FUNCTION_BLOCK FB_EmpujarPlato_SFC

VAR_IN_OUT
	   TpoEmpujadorAvanza: TIME;
END_VAR

VAR_INPUT
    // SFC-Flags
    SFCPause: BOOL;
    SFCReset: BOOL;
    
    // Indicadores de sincronizacion
    Ack: BOOL := TRUE;
    Execute: BOOL;
    
    
    // Entradas
   PlatoEmpujadorDetras : BOOL;
END_VAR
VAR_OUTPUT
    // Indicadores de sincronizacion
    Done: BOOL;
    Ready: BOOL;
    
    // Salidas
    PlatoEmpujadorAvanza : BOOL;
	PlatoRetenedorAtras : BOOL;
END_VAR
VAR
END_VAR

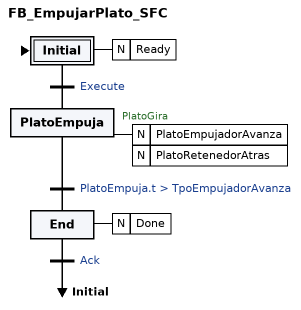
INITIAL_STEP Initial:
    Ready(N);
END_STEP
TRANSITION FROM Initial TO PlatoEmpuja
    := Execute;
END_TRANSITION
// PlatoGira
STEP PlatoEmpuja:
    PlatoEmpujadorAvanza(N);
    PlatoRetenedorAtras(N);
END_STEP
TRANSITION FROM PlatoEmpuja TO End
    := PlatoEmpuja.t > TpoEmpujadorAvanza;
END_TRANSITION
STEP End:
    Done(N);
END_STEP
TRANSITION FROM End TO Initial
    := Ack;
END_TRANSITION

END_FUNCTION_BLOCK

(* stored: Version 1.1.0.1, ProductVersion 3.1.4024.9
   POU FB_EmpujarPlato_SFC: Id {f8a809f5-43a3-4ce4-8569-3fd5eddc0b07}, SpecialFunc None *)
